Staubli VAL3: Pick.pgx

program Pick(pointRx pPos)
begin
end
